LIN {X 0,Y 105.585,Z 420.794,A -85,B 0,C 180,E1 -28240.561,E2 -28240.561} C_VEL
LIN {X 0,Y 105.28,Z 416.678,A -85,B 0,C 180,E1 -28246.489,E2 -28246.489} C_VEL
LIN {X 0,Y 105.21,Z 415.528,A -85,B 0,C 180,E1 -28248.44,E2 -28248.44} C_VEL
LIN {X 0,Y 104.972,Z 413.913,A -85,B 0,C 180,E1 -28252.305,E2 -28252.305} C_VEL
LIN {X 0,Y 105.02,Z 412.014,A -85,B 0,C 180,E1 -28260,E2 -28260} C_VEL
LIN {X 0,Y 104.682,Z 413.549,A -85,B 0,C 180,E1 -28267.965,E2 -28267.965} C_VEL
LIN {X 0,Y 104.931,Z 414.64,A -85,B 0,C 180,E1 -28271.592,E2 -28271.592} C_VEL
LIN {X 0,Y 105.458,Z 417.344,A -85,B 0,C 180,E1 -28277.451,E2 -28277.451} C_VEL
LIN {X 0,Y 106.084,Z 421.23,A -85,B 0,C 180,E1 -28283.422,E2 -28283.422} C_VEL
LIN {X 0,Y 106.272,Z 422.814,A -85,B 0,C 180,E1 -28285.459,E2 -28285.459} C_VEL
LIN {X 0,Y 106.144,Z 427.761,A -85,B 0,C 180,E1 -28290.604,E2 -28290.604} C_VEL
LIN {X 0,Y 105.861,Z 430.108,A -85,B 0,C 180,E1 -28292.818,E2 -28292.818} C_VEL
LIN {X 0,Y 104.957,Z 433.246,A -85,B 0,C 180,E1 -28295.32,E2 -28295.32} C_VEL
LIN {X 0,Y 103.734,Z 435.985,A -85,B 0,C 180,E1 -28297.247,E2 -28297.247} C_VEL
LIN {X 0,Y 96.488,Z 444.212,A -85,B 0,C 180,E1 -28301.708,E2 -28301.708} C_VEL
LIN {X 0,Y 90.783,Z 449.84,A -85,B 0,C 180,E1 -28305.838,E2 -28305.838} C_VEL
LIN {X 0,Y 84.545,Z 455.327,A -85,B 0,C 180,E1 -28311.435,E2 -28311.435} C_VEL
LIN {X 0,Y 79.313,Z 459.625,A -85,B 0,C 180,E1 -28317.885,E2 -28317.885} C_VEL
LIN {X 0,Y 76.364,Z 461.899,A -85,B 0,C 180,E1 -28322.605,E2 -28322.605} C_VEL
LIN {X 0,Y 73.924,Z 463.744,A -85,B 0,C 180,E1 -28327.652,E2 -28327.652} C_VEL
LIN {X 0,Y 70.79,Z 466.108,A -85,B 0,C 180,E1 -28338.55,E2 -28338.55} C_VEL
LIN {X 0,Y 70.624,Z 466.202,A -85,B 0,C 180,E1 -28339.423,E2 -28339.423} C_VEL
LIN {X 0,Y 69.303,Z 466.738,A -85,B 0,C 180,E1 -28344.127,E2 -28344.127} C_VEL
LIN {X 0,Y 66.179,Z 467,A -85,B 0,C 180,E1 -28352.101,E2 -28352.101} C_VEL
LIN {X 0,Y 64.321,Z 466.717,A -85,B 0,C 180,E1 -28358.943,E2 -28358.943} C_VEL
LIN {X 0,Y 64.206,Z 466.166,A -85,B 0,C 180,E1 -28364.243,E2 -28364.243} C_VEL
LIN {X 0,Y 64.524,Z 465.854,A -85,B 0,C 180,E1 -28365.977,E2 -28365.977} C_VEL
LIN {X 0,Y 67.396,Z 464.039,A -85,B 0,C 180,E1 -28374.655,E2 -28374.655} C_VEL
LIN {X 0,Y 71.623,Z 461.169,A -85,B 0,C 180,E1 -28382.664,E2 -28382.664} C_VEL
LIN {X 0,Y 76.993,Z 457.275,A -85,B 0,C 180,E1 -28389.717,E2 -28389.717} C_VEL
LIN {X 0,Y 83.457,Z 452.243,A -85,B 0,C 180,E1 -28395.71,E2 -28395.71} C_VEL
LIN {X 0,Y 90.599,Z 445.904,A -85,B 0,C 180,E1 -28400.873,E2 -28400.873} C_VEL
LIN {X 0,Y 98.238,Z 437.984,A -85,B 0,C 180,E1 -28405.355,E2 -28405.355} C_VEL
LIN {X 0,Y 99.183,Z 436.524,A -85,B 0,C 180,E1 -28406.365,E2 -28406.365} C_VEL
LIN {X 0,Y 99.882,Z 435,A -85,B 0,C 180,E1 -28407.605,E2 -28407.605} C_VEL
LIN {X 0,Y 100.73,Z 431.797,A -85,B 0,C 180,E1 -28410.765,E2 -28410.765} C_VEL
LIN {X 0,Y 101.227,Z 427.772,A -85,B 0,C 180,E1 -28415.382,E2 -28415.382} C_VEL
LIN {X 0,Y 101.117,Z 424.887,A -85,B 0,C 180,E1 -28419.664,E2 -28419.664} C_VEL
LIN {X 0,Y 100.898,Z 422.607,A -85,B 0,C 180,E1 -28423.822,E2 -28423.822} C_VEL
LIN {X 0,Y 100.756,Z 420.842,A -85,B 0,C 180,E1 -28427.921,E2 -28427.921} C_VEL
LIN {X 0,Y 100.642,Z 419.585,A -85,B 0,C 180,E1 -28431.971,E2 -28431.971} C_VEL
LIN {X 0,Y 100.984,Z 418.229,A -85,B 0,C 180,E1 -28440,E2 -28440} C_VEL
LIN {X 0,Y 100.887,Z 420.092,A -85,B 0,C 180,E1 -28448.009,E2 -28448.009} C_VEL
LIN {X 0,Y 100.936,Z 422.857,A -85,B 0,C 180,E1 -28453.899,E2 -28453.899} C_VEL
LIN {X 0,Y 100.864,Z 425.757,A -85,B 0,C 180,E1 -28458.273,E2 -28458.273} C_VEL
LIN {X 0,Y 100.339,Z 430.991,A -85,B 0,C 180,E1 -28464.417,E2 -28464.417} C_VEL
LIN {X 0,Y 99.403,Z 436.189,A -85,B 0,C 180,E1 -28469.664,E2 -28469.664} C_VEL
LIN {X 0,Y 95.514,Z 442.743,A -85,B 0,C 180,E1 -28474.126,E2 -28474.126} C_VEL
LIN {X 0,Y 93.261,Z 445.496,A -85,B 0,C 180,E1 -28475.893,E2 -28475.893} C_VEL
LIN {X 0,Y 85.82,Z 452.677,A -85,B 0,C 180,E1 -28480.754,E2 -28480.754} C_VEL
LIN {X 0,Y 77.996,Z 459.22,A -85,B 0,C 180,E1 -28487.481,E2 -28487.481} C_VEL
LIN {X 0,Y 72.243,Z 463.553,A -85,B 0,C 180,E1 -28494.287,E2 -28494.287} C_VEL
LIN {X 0,Y 69,Z 465.849,A -85,B 0,C 180,E1 -28499.382,E2 -28499.382} C_VEL
LIN {X 0,Y 66.446,Z 467.713,A -85,B 0,C 180,E1 -28504.968,E2 -28504.968} C_VEL
LIN {X 0,Y 63.235,Z 470.118,A -85,B 0,C 180,E1 -28517.154,E2 -28517.154} C_VEL
LIN {X 0,Y 62.585,Z 470.732,A -85,B 0,C 180,E1 -28523.55,E2 -28523.55} C_VEL
LIN {X 0,Y 62.61,Z 470.951,A -85,B 0,C 180,E1 -28529.997,E2 -28529.997} C_VEL
LIN {X 0,Y 62.585,Z 470.716,A -85,B 0,C 180,E1 -28536.445,E2 -28536.445} C_VEL
LIN {X 0,Y 63.234,Z 470.091,A -85,B 0,C 180,E1 -28542.84,E2 -28542.84} C_VEL
LIN {X 0,Y 64.513,Z 469.077,A -85,B 0,C 180,E1 -28549.072,E2 -28549.072} C_VEL
LIN {X 0,Y 66.444,Z 467.659,A -85,B 0,C 180,E1 -28555.027,E2 -28555.027} C_VEL
LIN {X 0,Y 70.563,Z 464.699,A -85,B 0,C 180,E1 -28563.212,E2 -28563.212} C_VEL
LIN {X 0,Y 75.926,Z 460.702,A -85,B 0,C 180,E1 -28570.383,E2 -28570.383} C_VEL
LIN {X 0,Y 83.229,Z 454.761,A -85,B 0,C 180,E1 -28577.284,E2 -28577.284} C_VEL
LIN {X 0,Y 90.652,Z 447.865,A -85,B 0,C 180,E1 -28582.618,E2 -28582.618} C_VEL
LIN {X 0,Y 94.453,Z 443.931,A -85,B 0,C 180,E1 -28584.928,E2 -28584.928} C_VEL
LIN {X 0,Y 98.326,Z 437.876,A -85,B 0,C 180,E1 -28589.055,E2 -28589.055} C_VEL
LIN {X 0,Y 99.315,Z 436.035,A -85,B 0,C 180,E1 -28590.307,E2 -28590.307} C_VEL
LIN {X 0,Y 100.027,Z 432.312,A -85,B 0,C 180,E1 -28593.952,E2 -28593.952} C_VEL
LIN {X 0,Y 100.458,Z 428.924,A -85,B 0,C 180,E1 -28597.597,E2 -28597.597} C_VEL
LIN {X 0,Y 100.743,Z 425.567,A -85,B 0,C 180,E1 -28601.704,E2 -28601.704} C_VEL
LIN {X 0,Y 100.815,Z 421.66,A -85,B 0,C 180,E1 -28607.928,E2 -28607.928} C_VEL
LIN {X 0,Y 100.741,Z 419.889,A -85,B 0,C 180,E1 -28611.98,E2 -28611.98} C_VEL
LIN {X 0,Y 100.924,Z 417.894,A -85,B 0,C 180,E1 -28620,E2 -28620} C_VEL
LIN {X 0,Y 100.487,Z 419.363,A -85,B 0,C 180,E1 -28628.041,E2 -28628.041} C_VEL
LIN {X 0,Y 100.602,Z 420.632,A -85,B 0,C 180,E1 -28632.098,E2 -28632.098} C_VEL
LIN {X 0,Y 100.922,Z 423.386,A -85,B 0,C 180,E1 -28638.263,E2 -28638.263} C_VEL
LIN {X 0,Y 101.083,Z 426.242,A -85,B 0,C 180,E1 -28642.868,E2 -28642.868} C_VEL
LIN {X 0,Y 100.911,Z 429.439,A -85,B 0,C 180,E1 -28646.915,E2 -28646.915} C_VEL
LIN {X 0,Y 100.396,Z 432.935,A -85,B 0,C 180,E1 -28650.746,E2 -28650.746} C_VEL
LIN {X 0,Y 99.186,Z 436.228,A -85,B 0,C 180,E1 -28653.644,E2 -28653.644} C_VEL
LIN {X 0,Y 98.273,Z 437.685,A -85,B 0,C 180,E1 -28654.68,E2 -28654.68} C_VEL
LIN {X 0,Y 90.653,Z 445.655,A -85,B 0,C 180,E1 -28659.176,E2 -28659.176} C_VEL
LIN {X 0,Y 83.507,Z 452.053,A -85,B 0,C 180,E1 -28664.331,E2 -28664.331} C_VEL
LIN {X 0,Y 77.058,Z 457.127,A -85,B 0,C 180,E1 -28670.329,E2 -28670.329} C_VEL
LIN {X 0,Y 71.68,Z 461.059,A -85,B 0,C 180,E1 -28677.37,E2 -28677.37} C_VEL
LIN {X 0,Y 67.406,Z 463.961,A -85,B 0,C 180,E1 -28685.355,E2 -28685.355} C_VEL
LIN {X 0,Y 65.316,Z 465.342,A -85,B 0,C 180,E1 -28691.171,E2 -28691.171} C_VEL
LIN {X 0,Y 63.606,Z 466.441,A -85,B 0,C 180,E1 -28698.488,E2 -28698.488} C_VEL
LIN {X 0,Y 62.755,Z 467.146,A -85,B 0,C 180,E1 -28710.003,E2 -28710.003} C_VEL
LIN {X 0,Y 62.952,Z 466.95,A -85,B 0,C 180,E1 -28716.413,E2 -28716.413} C_VEL
LIN {X 0,Y 64.524,Z 465.854,A -85,B 0,C 180,E1 -28725.977,E2 -28725.977} C_VEL
LIN {X 0,Y 65.342,Z 465.002,A -85,B 0,C 180,E1 -28731.081,E2 -28731.081} C_VEL
LIN {X 0,Y 65.948,Z 463.074,A -85,B 0,C 180,E1 -28739.571,E2 -28739.571} C_VEL
LIN {X 0,Y 67.18,Z 461.056,A -85,B 0,C 180,E1 -28746.126,E2 -28746.126} C_VEL
LIN {X 0,Y 69.265,Z 459.175,A -85,B 0,C 180,E1 -28750.51,E2 -28750.51} C_VEL
LIN {X 0,Y 70.251,Z 458.446,A -85,B 0,C 180,E1 -28751.79,E2 -28751.79} C_VEL
LIN {X 0,Y 78.665,Z 452.457,A -85,B 0,C 180,E1 -28759.413,E2 -28759.413} C_VEL
LIN {X 0,Y 86.287,Z 446.117,A -85,B 0,C 180,E1 -28764.539,E2 -28764.539} C_VEL
LIN {X 0,Y 93.009,Z 439.668,A -85,B 0,C 180,E1 -28768.218,E2 -28768.218} C_VEL
LIN {X 0,Y 94.058,Z 438.215,A -85,B 0,C 180,E1 -28769.233,E2 -28769.233} C_VEL
LIN {X 0,Y 95.177,Z 435.281,A -85,B 0,C 180,E1 -28772.388,E2 -28772.388} C_VEL
LIN {X 0,Y 95.877,Z 432.272,A -85,B 0,C 180,E1 -28776.224,E2 -28776.224} C_VEL
LIN {X 0,Y 95.995,Z 430.765,A -85,B 0,C 180,E1 -28778.527,E2 -28778.527} C_VEL
LIN {X 0,Y 96.055,Z 428.389,A -85,B 0,C 180,E1 -28782.982,E2 -28782.982} C_VEL
LIN {X 0,Y 96.039,Z 426.549,A -85,B 0,C 180,E1 -28787.318,E2 -28787.318} C_VEL
LIN {X 0,Y 96.1,Z 425.235,A -85,B 0,C 180,E1 -28791.589,E2 -28791.589} C_VEL
LIN {X 0,Y 96.563,Z 423.859,A -85,B 0,C 180,E1 -28800,E2 -28800} C_VEL
LIN {X 0,Y 96.326,Z 424.669,A -85,B 0,C 180,E1 -28804.184,E2 -28804.184} C_VEL
LIN {X 0,Y 96.282,Z 425.864,A -85,B 0,C 180,E1 -28808.394,E2 -28808.394} C_VEL
LIN {X 0,Y 96.145,Z 427.688,A -85,B 0,C 180,E1 -28812.667,E2 -28812.667} C_VEL
LIN {X 0,Y 95.774,Z 430.609,A -85,B 0,C 180,E1 -28817.452,E2 -28817.452} C_VEL
LIN {X 0,Y 94.924,Z 434.889,A -85,B 0,C 180,E1 -28822.993,E2 -28822.993} C_VEL
LIN {X 0,Y 94.095,Z 438.07,A -85,B 0,C 180,E1 -28826.625,E2 -28826.625} C_VEL
LIN {X 0,Y 93.37,Z 439.657,A -85,B 0,C 180,E1 -28828.078,E2 -28828.078} C_VEL
LIN {X 0,Y 89.232,Z 445.28,A -85,B 0,C 180,E1 -28832.146,E2 -28832.146} C_VEL
LIN {X 0,Y 81.339,Z 452.462,A -85,B 0,C 180,E1 -28836.941,E2 -28836.941} C_VEL
LIN {X 0,Y 75.244,Z 457.315,A -85,B 0,C 180,E1 -28841.648,E2 -28841.648} C_VEL
LIN {X 0,Y 68.582,Z 462.029,A -85,B 0,C 180,E1 -28848.231,E2 -28848.231} C_VEL
LIN {X 0,Y 62.974,Z 465.634,A -85,B 0,C 180,E1 -28856.079,E2 -28856.079} C_VEL
LIN {X 0,Y 60.046,Z 467.497,A -85,B 0,C 180,E1 -28862.081,E2 -28862.081} C_VEL
LIN {X 0,Y 57.837,Z 468.899,A -85,B 0,C 180,E1 -28868.618,E2 -28868.618} C_VEL
LIN {X 0,Y 56.317,Z 469.902,A -85,B 0,C 180,E1 -28875.544,E2 -28875.544} C_VEL
LIN {X 0,Y 55.54,Z 470.517,A -85,B 0,C 180,E1 -28882.727,E2 -28882.727} C_VEL
LIN {X 0,Y 55.509,Z 470.736,A -85,B 0,C 180,E1 -28889.997,E2 -28889.997} C_VEL
LIN {X 0,Y 55.539,Z 470.5,A -85,B 0,C 180,E1 -28897.266,E2 -28897.266} C_VEL
LIN {X 0,Y 56.315,Z 469.875,A -85,B 0,C 180,E1 -28904.45,E2 -28904.45} C_VEL
LIN {X 0,Y 57.835,Z 468.86,A -85,B 0,C 180,E1 -28911.376,E2 -28911.376} C_VEL
LIN {X 0,Y 60.043,Z 467.442,A -85,B 0,C 180,E1 -28917.913,E2 -28917.913} C_VEL
LIN {X 0,Y 64.724,Z 464.482,A -85,B 0,C 180,E1 -28926.666,E2 -28926.666} C_VEL
LIN {X 0,Y 70.648,Z 460.485,A -85,B 0,C 180,E1 -28934.13,E2 -28934.13} C_VEL
LIN {X 0,Y 77.893,Z 455.091,A -85,B 0,C 180,E1 -28940.609,E2 -28940.609} C_VEL
LIN {X 0,Y 86.502,Z 447.646,A -85,B 0,C 180,E1 -28946.38,E2 -28946.38} C_VEL
LIN {X 0,Y 89.2,Z 445.075,A -85,B 0,C 180,E1 -28947.88,E2 -28947.88} C_VEL
LIN {X 0,Y 93.317,Z 439.465,A -85,B 0,C 180,E1 -28951.922,E2 -28951.922} C_VEL
LIN {X 0,Y 94.117,Z 437.606,A -85,B 0,C 180,E1 -28953.641,E2 -28953.641} C_VEL
LIN {X 0,Y 95.06,Z 433.603,A -85,B 0,C 180,E1 -28958.305,E2 -28958.305} C_VEL
LIN {X 0,Y 95.726,Z 430.132,A -85,B 0,C 180,E1 -28962.922,E2 -28962.922} C_VEL
LIN {X 0,Y 96.017,Z 427.508,A -85,B 0,C 180,E1 -28967.315,E2 -28967.315} C_VEL
LIN {X 0,Y 96.162,Z 425.655,A -85,B 0,C 180,E1 -28971.595,E2 -28971.595} C_VEL
LIN {X 0,Y 96.225,Z 424.422,A -85,B 0,C 180,E1 -28975.812,E2 -28975.812} C_VEL
LIN {X 0,Y 96.517,Z 423.536,A -85,B 0,C 180,E1 -28980,E2 -28980} C_VEL
LIN {X 0,Y 95.947,Z 425.044,A -85,B 0,C 180,E1 -28988.424,E2 -28988.424} C_VEL
LIN {X 0,Y 95.912,Z 426.328,A -85,B 0,C 180,E1 -28992.699,E2 -28992.699} C_VEL
LIN {X 0,Y 95.974,Z 429.117,A -85,B 0,C 180,E1 -28999.018,E2 -28999.018} C_VEL
LIN {X 0,Y 95.757,Z 432.06,A -85,B 0,C 180,E1 -29003.808,E2 -29003.808} C_VEL
LIN {X 0,Y 95.126,Z 434.969,A -85,B 0,C 180,E1 -29007.561,E2 -29007.561} C_VEL
LIN {X 0,Y 94.705,Z 436.493,A -85,B 0,C 180,E1 -29009.323,E2 -29009.323} C_VEL
LIN {X 0,Y 94.055,Z 437.924,A -85,B 0,C 180,E1 -29010.771,E2 -29010.771} C_VEL
LIN {X 0,Y 93.043,Z 439.38,A -85,B 0,C 180,E1 -29011.823,E2 -29011.823} C_VEL
LIN {X 0,Y 85.048,Z 447.033,A -85,B 0,C 180,E1 -29016.327,E2 -29016.327} C_VEL
LIN {X 0,Y 76.307,Z 454.074,A -85,B 0,C 180,E1 -29022.544,E2 -29022.544} C_VEL
LIN {X 0,Y 69.669,Z 458.756,A -85,B 0,C 180,E1 -29029.032,E2 -29029.032} C_VEL
LIN {X 0,Y 64.072,Z 462.333,A -85,B 0,C 180,E1 -29036.744,E2 -29036.744} C_VEL
LIN {X 0,Y 61.027,Z 464.177,A -85,B 0,C 180,E1 -29042.575,E2 -29042.575} C_VEL
LIN {X 0,Y 58.634,Z 465.558,A -85,B 0,C 180,E1 -29048.929,E2 -29048.929} C_VEL
LIN {X 0,Y 56.927,Z 466.54,A -85,B 0,C 180,E1 -29055.709,E2 -29055.709} C_VEL
LIN {X 0,Y 55.671,Z 467.361,A -85,B 0,C 180,E1 -29070.003,E2 -29070.003} C_VEL
LIN {X 0,Y 55.92,Z 467.165,A -85,B 0,C 180,E1 -29077.223,E2 -29077.223} C_VEL
LIN {X 0,Y 57.623,Z 466.127,A -85,B 0,C 180,E1 -29087.514,E2 -29087.514} C_VEL
LIN {X 0,Y 61.015,Z 464.253,A -85,B 0,C 180,E1 -29097.437,E2 -29097.437} C_VEL
LIN {X 0,Y 65.755,Z 461.384,A -85,B 0,C 180,E1 -29106.007,E2 -29106.007} C_VEL
LIN {X 0,Y 70.251,Z 458.446,A -85,B 0,C 180,E1 -29111.79,E2 -29111.79} C_VEL
LIN {X 0,Y 73.05,Z 456.216,A -85,B 0,C 180,E1 -29115.557,E2 -29115.557} C_VEL
LIN {X 0,Y 76.861,Z 452.182,A -85,B 0,C 180,E1 -29121.862,E2 -29121.862} C_VEL
LIN {X 0,Y 81.242,Z 447.528,A -85,B 0,C 180,E1 -29127.366,E2 -29127.366} C_VEL
LIN {X 0,Y 84.73,Z 444.272,A -85,B 0,C 180,E1 -29129.795,E2 -29129.795} C_VEL
LIN {X 0,Y 88.036,Z 441.237,A -85,B 0,C 180,E1 -29131.421,E2 -29131.421} C_VEL
LIN {X 0,Y 89.108,Z 439.823,A -85,B 0,C 180,E1 -29132.684,E2 -29132.684} C_VEL
LIN {X 0,Y 90.314,Z 436.591,A -85,B 0,C 180,E1 -29137.102,E2 -29137.102} C_VEL
LIN {X 0,Y 90.779,Z 433.928,A -85,B 0,C 180,E1 -29141.96,E2 -29141.96} C_VEL
LIN {X 0,Y 90.981,Z 432.024,A -85,B 0,C 180,E1 -29146.6,E2 -29146.6} C_VEL
LIN {X 0,Y 91.175,Z 430.632,A -85,B 0,C 180,E1 -29151.131,E2 -29151.131} C_VEL
LIN {X 0,Y 91.507,Z 429.598,A -85,B 0,C 180,E1 -29156.807,E2 -29156.807} C_VEL
LIN {X 0,Y 91.845,Z 429.233,A -85,B 0,C 180,E1 -29160,E2 -29160} C_VEL
LIN {X 0,Y 91.535,Z 430.065,A -85,B 0,C 180,E1 -29164.403,E2 -29164.403} C_VEL
LIN {X 0,Y 91.154,Z 432.227,A -85,B 0,C 180,E1 -29171.113,E2 -29171.113} C_VEL
LIN {X 0,Y 90.648,Z 434.644,A -85,B 0,C 180,E1 -29175.745,E2 -29175.745} C_VEL
LIN {X 0,Y 89.379,Z 438.718,A -85,B 0,C 180,E1 -29181.607,E2 -29181.607} C_VEL
LIN {X 0,Y 88.28,Z 441.474,A -85,B 0,C 180,E1 -29185.018,E2 -29185.018} C_VEL
LIN {X 0,Y 85.479,Z 445.055,A -85,B 0,C 180,E1 -29187.886,E2 -29187.886} C_VEL
LIN {X 0,Y 82.814,Z 447.619,A -85,B 0,C 180,E1 -29189.554,E2 -29189.554} C_VEL
LIN {X 0,Y 74.429,Z 454.377,A -85,B 0,C 180,E1 -29194.51,E2 -29194.51} C_VEL
LIN {X 0,Y 65.73,Z 460.377,A -85,B 0,C 180,E1 -29201.54,E2 -29201.54} C_VEL
LIN {X 0,Y 59.174,Z 464.345,A -85,B 0,C 180,E1 -29209.212,E2 -29209.212} C_VEL
LIN {X 0,Y 53.836,Z 467.281,A -85,B 0,C 180,E1 -29218.519,E2 -29218.519} C_VEL
LIN {X 0,Y 49.467,Z 469.687,A -85,B 0,C 180,E1 -29233.488,E2 -29233.488} C_VEL
LIN {X 0,Y 48.497,Z 470.302,A -85,B 0,C 180,E1 -29241.664,E2 -29241.664} C_VEL
LIN {X 0,Y 48.427,Z 470.521,A -85,B 0,C 180,E1 -29249.996,E2 -29249.996} C_VEL
LIN {X 0,Y 48.496,Z 470.284,A -85,B 0,C 180,E1 -29258.329,E2 -29258.329} C_VEL
LIN {X 0,Y 49.465,Z 469.659,A -85,B 0,C 180,E1 -29266.505,E2 -29266.505} C_VEL
LIN {X 0,Y 51.248,Z 468.643,A -85,B 0,C 180,E1 -29274.289,E2 -29274.289} C_VEL
LIN {X 0,Y 53.833,Z 467.224,A -85,B 0,C 180,E1 -29281.476,E2 -29281.476} C_VEL
LIN {X 0,Y 59.17,Z 464.265,A -85,B 0,C 180,E1 -29290.784,E2 -29290.784} C_VEL
LIN {X 0,Y 65.724,Z 460.267,A -85,B 0,C 180,E1 -29298.457,E2 -29298.457} C_VEL
LIN {X 0,Y 74.36,Z 454.268,A -85,B 0,C 180,E1 -29305.454,E2 -29305.454} C_VEL
LIN {X 0,Y 82.771,Z 447.428,A -85,B 0,C 180,E1 -29310.489,E2 -29310.489} C_VEL
LIN {X 0,Y 85.44,Z 444.844,A -85,B 0,C 180,E1 -29312.153,E2 -29312.153} C_VEL
LIN {X 0,Y 88.214,Z 441.319,A -85,B 0,C 180,E1 -29314.929,E2 -29314.929} C_VEL
LIN {X 0,Y 89.684,Z 437.26,A -85,B 0,C 180,E1 -29320.104,E2 -29320.104} C_VEL
LIN {X 0,Y 90.589,Z 434.147,A -85,B 0,C 180,E1 -29324.849,E2 -29324.849} C_VEL
LIN {X 0,Y 91.034,Z 432.053,A -85,B 0,C 180,E1 -29328.872,E2 -29328.872} C_VEL
LIN {X 0,Y 91.186,Z 431.16,A -85,B 0,C 180,E1 -29331.133,E2 -29331.133} C_VEL
LIN {X 0,Y 91.521,Z 429.594,A -85,B 0,C 180,E1 -29336.589,E2 -29336.589} C_VEL
LIN {X 0,Y 91.814,Z 428.923,A -85,B 0,C 180,E1 -29340,E2 -29340} C_VEL
LIN {X 0,Y 91.037,Z 430.448,A -85,B 0,C 180,E1 -29348.882,E2 -29348.882} C_VEL
LIN {X 0,Y 90.879,Z 431.799,A -85,B 0,C 180,E1 -29353.415,E2 -29353.415} C_VEL
LIN {X 0,Y 90.744,Z 433.654,A -85,B 0,C 180,E1 -29358.047,E2 -29358.047} C_VEL
LIN {X 0,Y 90.219,Z 436.382,A -85,B 0,C 180,E1 -29362.924,E2 -29362.924} C_VEL
LIN {X 0,Y 89.013,Z 439.744,A -85,B 0,C 180,E1 -29367.562,E2 -29367.562} C_VEL
LIN {X 0,Y 88.076,Z 440.972,A -85,B 0,C 180,E1 -29368.635,E2 -29368.635} C_VEL
LIN {X 0,Y 79.69,Z 448.359,A -85,B 0,C 180,E1 -29373.095,E2 -29373.095} C_VEL
LIN {X 0,Y 71.689,Z 454.291,A -85,B 0,C 180,E1 -29378.352,E2 -29378.352} C_VEL
LIN {X 0,Y 64.458,Z 458.973,A -85,B 0,C 180,E1 -29384.875,E2 -29384.875} C_VEL
LIN {X 0,Y 58.254,Z 462.549,A -85,B 0,C 180,E1 -29392.904,E2 -29392.904} C_VEL
LIN {X 0,Y 54.83,Z 464.393,A -85,B 0,C 180,E1 -29399.16,E2 -29399.16} C_VEL
LIN {X 0,Y 52.076,Z 465.774,A -85,B 0,C 180,E1 -29406.121,E2 -29406.121} C_VEL
LIN {X 0,Y 50.085,Z 466.756,A -85,B 0,C 180,E1 -29413.705,E2 -29413.705} C_VEL
LIN {X 0,Y 48.581,Z 467.577,A -85,B 0,C 180,E1 -29430.004,E2 -29430.004} C_VEL
LIN {X 0,Y 48.885,Z 467.38,A -85,B 0,C 180,E1 -29438.269,E2 -29438.269} C_VEL
LIN {X 0,Y 50.086,Z 466.793,A -85,B 0,C 180,E1 -29446.302,E2 -29446.302} C_VEL
LIN {X 0,Y 54.817,Z 464.468,A -85,B 0,C 180,E1 -29460.856,E2 -29460.856} C_VEL
LIN {X 0,Y 60.155,Z 461.598,A -85,B 0,C 180,E1 -29469.987,E2 -29469.987} C_VEL
LIN {X 0,Y 66.683,Z 457.704,A -85,B 0,C 180,E1 -29477.544,E2 -29477.544} C_VEL
LIN {X 0,Y 74.244,Z 452.67,A -85,B 0,C 180,E1 -29483.576,E2 -29483.576} C_VEL
LIN {X 0,Y 82.368,Z 446.331,A -85,B 0,C 180,E1 -29488.569,E2 -29488.569} C_VEL
LIN {X 0,Y 84.73,Z 444.272,A -85,B 0,C 180,E1 -29489.795,E2 -29489.795} C_VEL
LIN {X 0,Y 85.953,Z 442.94,A -85,B 0,C 180,E1 -29490.916,E2 -29490.916} C_VEL
LIN {X 0,Y 86.622,Z 441.391,A -85,B 0,C 180,E1 -29493.19,E2 -29493.19} C_VEL
LIN {X 0,Y 86.42,Z 440.352,A -85,B 0,C 180,E1 -29495.719,E2 -29495.719} C_VEL
LIN {X 0,Y 85.262,Z 438.124,A -85,B 0,C 180,E1 -29503.569,E2 -29503.569} C_VEL
LIN {X 0,Y 85.826,Z 436.126,A -85,B 0,C 180,E1 -29509.314,E2 -29509.314} C_VEL
LIN {X 0,Y 86.279,Z 434.86,A -85,B 0,C 180,E1 -29515.327,E2 -29515.327} C_VEL
LIN {X 0,Y 86.813,Z 434.311,A -85,B 0,C 180,E1 -29520,E2 -29520} C_VEL
LIN {X 0,Y 86.366,Z 435.2,A -85,B 0,C 180,E1 -29524.667,E2 -29524.667} C_VEL
LIN {X 0,Y 85.841,Z 437.082,A -85,B 0,C 180,E1 -29530.738,E2 -29530.738} C_VEL
LIN {X 0,Y 85.292,Z 438.748,A -85,B 0,C 180,E1 -29534.312,E2 -29534.312} C_VEL
LIN {X 0,Y 83.883,Z 442.007,A -85,B 0,C 180,E1 -29539.581,E2 -29539.581} C_VEL
LIN {X 0,Y 83.159,Z 443.421,A -85,B 0,C 180,E1 -29541.619,E2 -29541.619} C_VEL
LIN {X 0,Y 82.159,Z 444.824,A -85,B 0,C 180,E1 -29543.133,E2 -29543.133} C_VEL
LIN {X 0,Y 79.538,Z 447.404,A -85,B 0,C 180,E1 -29545.081,E2 -29545.081} C_VEL
LIN {X 0,Y 69.862,Z 454.709,A -85,B 0,C 180,E1 -29550.198,E2 -29550.198} C_VEL
LIN {X 0,Y 61.243,Z 460.163,A -85,B 0,C 180,E1 -29556.551,E2 -29556.551} C_VEL
LIN {X 0,Y 53.97,Z 464.129,A -85,B 0,C 180,E1 -29564.253,E2 -29564.253} C_VEL
LIN {X 0,Y 47.891,Z 467.065,A -85,B 0,C 180,E1 -29574.052,E2 -29574.052} C_VEL
LIN {X 0,Y 42.676,Z 469.471,A -85,B 0,C 180,E1 -29590.766,E2 -29590.766} C_VEL
LIN {X 0,Y 41.471,Z 470.086,A -85,B 0,C 180,E1 -29600.239,E2 -29600.239} C_VEL
LIN {X 0,Y 41.327,Z 470.305,A -85,B 0,C 180,E1 -29609.996,E2 -29609.996} C_VEL
LIN {X 0,Y 41.47,Z 470.068,A -85,B 0,C 180,E1 -29619.753,E2 -29619.753} C_VEL
LIN {X 0,Y 42.674,Z 469.442,A -85,B 0,C 180,E1 -29629.227,E2 -29629.227} C_VEL
LIN {X 0,Y 44.834,Z 468.426,A -85,B 0,C 180,E1 -29638.047,E2 -29638.047} C_VEL
LIN {X 0,Y 47.888,Z 467.007,A -85,B 0,C 180,E1 -29645.942,E2 -29645.942} C_VEL
LIN {X 0,Y 53.965,Z 464.047,A -85,B 0,C 180,E1 -29655.742,E2 -29655.742} C_VEL
LIN {X 0,Y 61.237,Z 460.05,A -85,B 0,C 180,E1 -29663.447,E2 -29663.447} C_VEL
LIN {X 0,Y 69.933,Z 454.503,A -85,B 0,C 180,E1 -29669.836,E2 -29669.836} C_VEL
LIN {X 0,Y 79.494,Z 447.209,A -85,B 0,C 180,E1 -29674.978,E2 -29674.978} C_VEL
LIN {X 0,Y 82.133,Z 444.609,A -85,B 0,C 180,E1 -29676.898,E2 -29676.898} C_VEL
LIN {X 0,Y 83.112,Z 443.203,A -85,B 0,C 180,E1 -29678.452,E2 -29678.452} C_VEL
LIN {X 0,Y 84.492,Z 440.141,A -85,B 0,C 180,E1 -29683.075,E2 -29683.075} C_VEL
LIN {X 0,Y 85.131,Z 438.642,A -85,B 0,C 180,E1 -29685.661,E2 -29685.661} C_VEL
LIN {X 0,Y 85.89,Z 436.383,A -85,B 0,C 180,E1 -29690.581,E2 -29690.581} C_VEL
LIN {X 0,Y 86.291,Z 434.988,A -85,B 0,C 180,E1 -29695.329,E2 -29695.329} C_VEL
LIN {X 0,Y 86.799,Z 434.037,A -85,B 0,C 180,E1 -29700,E2 -29700} C_VEL
LIN {X 0,Y 85.859,Z 435.3,A -85,B 0,C 180,E1 -29707.904,E2 -29707.904} C_VEL
LIN {X 0,Y 85.475,Z 437.044,A -85,B 0,C 180,E1 -29714.281,E2 -29714.281} C_VEL
LIN {X 0,Y 85.34,Z 437.882,A -85,B 0,C 180,E1 -29716.753,E2 -29716.753} C_VEL
LIN {X 0,Y 84.727,Z 439.914,A -85,B 0,C 180,E1 -29720.99,E2 -29720.99} C_VEL
LIN {X 0,Y 83.595,Z 442.308,A -85,B 0,C 180,E1 -29724.858,E2 -29724.858} C_VEL
LIN {X 0,Y 74.61,Z 449.685,A -85,B 0,C 180,E1 -29729.395,E2 -29729.395} C_VEL
LIN {X 0,Y 67.511,Z 454.509,A -85,B 0,C 180,E1 -29733.617,E2 -29733.617} C_VEL
LIN {X 0,Y 59.65,Z 459.191,A -85,B 0,C 180,E1 -29740.025,E2 -29740.025} C_VEL
LIN {X 0,Y 52.761,Z 462.766,A -85,B 0,C 180,E1 -29748.245,E2 -29748.245} C_VEL
LIN {X 0,Y 48.856,Z 464.609,A -85,B 0,C 180,E1 -29754.878,E2 -29754.878} C_VEL
LIN {X 0,Y 43.334,Z 466.971,A -85,B 0,C 180,E1 -29771.078,E2 -29771.078} C_VEL
LIN {X 0,Y 41.481,Z 467.792,A -85,B 0,C 180,E1 -29790.004,E2 -29790.004} C_VEL
LIN {X 0,Y 41.888,Z 467.595,A -85,B 0,C 180,E1 -29799.663,E2 -29799.663} C_VEL
LIN {X 0,Y 43.336,Z 467.008,A -85,B 0,C 180,E1 -29808.93,E2 -29808.93} C_VEL
LIN {X 0,Y 48.843,Z 464.683,A -85,B 0,C 180,E1 -29825.143,E2 -29825.143} C_VEL
LIN {X 0,Y 54.906,Z 461.813,A -85,B 0,C 180,E1 -29834.753,E2 -29834.753} C_VEL
LIN {X 0,Y 62.113,Z 457.918,A -85,B 0,C 180,E1 -29842.38,E2 -29842.38} C_VEL
LIN {X 0,Y 70.264,Z 452.884,A -85,B 0,C 180,E1 -29848.235,E2 -29848.235} C_VEL
LIN {X 0,Y 78.898,Z 446.544,A -85,B 0,C 180,E1 -29852.973,E2 -29852.973} C_VEL
LIN {X 0,Y 83.617,Z 442.551,A -85,B 0,C 180,E1 -29855.149,E2 -29855.149} C_VEL
LIN {X 0,Y 84.791,Z 440.203,A -85,B 0,C 180,E1 -29858.861,E2 -29858.861} C_VEL
LIN {X 0,Y 85.079,Z 439.255,A -85,B 0,C 180,E1 -29860.705,E2 -29860.705} C_VEL
LIN {X 0,Y 85.262,Z 438.124,A -85,B 0,C 180,E1 -29863.569,E2 -29863.569} C_VEL
LIN {X 0,Y 84.964,Z 437.63,A -85,B 0,C 180,E1 -29866.166,E2 -29866.166} C_VEL
LIN {X 0,Y 83.546,Z 438.055,A -85,B 0,C 180,E1 -29869.64,E2 -29869.64} C_VEL
LIN {X 0,Y 81.319,Z 439.28,A -85,B 0,C 180,E1 -29875.09,E2 -29875.09} C_VEL
LIN {X 0,Y 81.147,Z 439.339,A -85,B 0,C 180,E1 -29877.969,E2 -29877.969} C_VEL
LIN {X 0,Y 81.474,Z 439.106,A -85,B 0,C 180,E1 -29880,E2 -29880} C_VEL
LIN {X 0,Y 80.898,Z 440.062,A -85,B 0,C 180,E1 -29884.984,E2 -29884.984} C_VEL
LIN {X 0,Y 80.304,Z 441.559,A -85,B 0,C 180,E1 -29890.08,E2 -29890.08} C_VEL
LIN {X 0,Y 79.521,Z 443.06,A -85,B 0,C 180,E1 -29893.543,E2 -29893.543} C_VEL
LIN {X 0,Y 77.856,Z 445.906,A -85,B 0,C 180,E1 -29898.586,E2 -29898.586} C_VEL
LIN {X 0,Y 76.709,Z 447.183,A -85,B 0,C 180,E1 -29900.096,E2 -29900.096} C_VEL
LIN {X 0,Y 69.051,Z 452.839,A -85,B 0,C 180,E1 -29903.645,E2 -29903.645} C_VEL
LIN {X 0,Y 60.168,Z 458.361,A -85,B 0,C 180,E1 -29908.827,E2 -29908.827} C_VEL
LIN {X 0,Y 51.845,Z 462.692,A -85,B 0,C 180,E1 -29915.571,E2 -29915.571} C_VEL
LIN {X 0,Y 46.804,Z 464.989,A -85,B 0,C 180,E1 -29921.336,E2 -29921.336} C_VEL
LIN {X 0,Y 42.32,Z 466.849,A -85,B 0,C 180,E1 -29928.369,E2 -29928.369} C_VEL
LIN {X 0,Y 36.027,Z 469.255,A -85,B 0,C 180,E1 -29947.031,E2 -29947.031} C_VEL
LIN {X 0,Y 34.493,Z 469.871,A -85,B 0,C 180,E1 -29958.238,E2 -29958.238} C_VEL
LIN {X 0,Y 34.242,Z 470.09,A -85,B 0,C 180,E1 -29969.995,E2 -29969.995} C_VEL
LIN {X 0,Y 34.491,Z 469.852,A -85,B 0,C 180,E1 -29981.751,E2 -29981.751} C_VEL
LIN {X 0,Y 36.025,Z 469.225,A -85,B 0,C 180,E1 -29992.96,E2 -29992.96} C_VEL
LIN {X 0,Y 38.684,Z 468.209,A -85,B 0,C 180,E1 -30003.021,E2 -30003.021} C_VEL
LIN {X 0,Y 42.316,Z 466.789,A -85,B 0,C 180,E1 -30011.625,E2 -30011.625} C_VEL
LIN {X 0,Y 49.254,Z 463.83,A -85,B 0,C 180,E1 -30021.694,E2 -30021.694} C_VEL
LIN {X 0,Y 57.287,Z 459.833,A -85,B 0,C 180,E1 -30029.17,E2 -30029.17} C_VEL
LIN {X 0,Y 67.462,Z 453.724,A -85,B 0,C 180,E1 -30035.595,E2 -30035.595} C_VEL
LIN {X 0,Y 76.679,Z 446.987,A -85,B 0,C 180,E1 -30039.944,E2 -30039.944} C_VEL
LIN {X 0,Y 77.814,Z 445.71,A -85,B 0,C 180,E1 -30041.477,E2 -30041.477} C_VEL
LIN {X 0,Y 79.454,Z 442.83,A -85,B 0,C 180,E1 -30046.638,E2 -30046.638} C_VEL
LIN {X 0,Y 80.176,Z 441.42,A -85,B 0,C 180,E1 -30049.903,E2 -30049.903} C_VEL
LIN {X 0,Y 80.82,Z 439.871,A -85,B 0,C 180,E1 -30055.012,E2 -30055.012} C_VEL
LIN {X 0,Y 81.457,Z 438.858,A -85,B 0,C 180,E1 -30060,E2 -30060} C_VEL
LIN {X 0,Y 80.438,Z 439.997,A -85,B 0,C 180,E1 -30067.665,E2 -30067.665} C_VEL
LIN {X 0,Y 80.287,Z 440.464,A -85,B 0,C 180,E1 -30070.083,E2 -30070.083} C_VEL
LIN {X 0,Y 79.777,Z 441.9,A -85,B 0,C 180,E1 -30075.325,E2 -30075.325} C_VEL
LIN {X 0,Y 79.354,Z 442.944,A -85,B 0,C 180,E1 -30078.058,E2 -30078.058} C_VEL
LIN {X 0,Y 78.591,Z 444.366,A -85,B 0,C 180,E1 -30080.959,E2 -30080.959} C_VEL
LIN {X 0,Y 77.371,Z 445.42,A -85,B 0,C 180,E1 -30081.751,E2 -30081.751} C_VEL
LIN {X 0,Y 69.845,Z 450.926,A -85,B 0,C 180,E1 -30085.103,E2 -30085.103} C_VEL
LIN {X 0,Y 60.948,Z 456.411,A -85,B 0,C 180,E1 -30090.143,E2 -30090.143} C_VEL
LIN {X 0,Y 52.685,Z 460.711,A -85,B 0,C 180,E1 -30096.841,E2 -30096.841} C_VEL
LIN {X 0,Y 47.701,Z 462.982,A -85,B 0,C 180,E1 -30102.558,E2 -30102.558} C_VEL
LIN {X 0,Y 43.237,Z 464.826,A -85,B 0,C 180,E1 -30109.451,E2 -30109.451} C_VEL
LIN {X 0,Y 36.694,Z 467.187,A -85,B 0,C 180,E1 -30127.483,E2 -30127.483} C_VEL
LIN {X 0,Y 34.4,Z 468.007,A -85,B 0,C 180,E1 -30150.005,E2 -30150.005} C_VEL
LIN {X 0,Y 34.92,Z 467.81,A -85,B 0,C 180,E1 -30161.616,E2 -30161.616} C_VEL
LIN {X 0,Y 36.696,Z 467.223,A -85,B 0,C 180,E1 -30172.527,E2 -30172.527} C_VEL
LIN {X 0,Y 43.224,Z 464.898,A -85,B 0,C 180,E1 -30190.575,E2 -30190.575} C_VEL
LIN {X 0,Y 50.115,Z 462.027,A -85,B 0,C 180,E1 -30200.476,E2 -30200.476} C_VEL
LIN {X 0,Y 58.056,Z 458.132,A -85,B 0,C 180,E1 -30207.933,E2 -30207.933} C_VEL
LIN {X 0,Y 66.803,Z 453.098,A -85,B 0,C 180,E1 -30213.414,E2 -30213.414} C_VEL
LIN {X 0,Y 75.937,Z 446.758,A -85,B 0,C 180,E1 -30217.748,E2 -30217.748} C_VEL
LIN {X 0,Y 78.629,Z 444.571,A -85,B 0,C 180,E1 -30219.051,E2 -30219.051} C_VEL
LIN {X 0,Y 79.405,Z 443.157,A -85,B 0,C 180,E1 -30221.954,E2 -30221.954} C_VEL
LIN {X 0,Y 80.393,Z 440.641,A -85,B 0,C 180,E1 -30229.93,E2 -30229.93} C_VEL
LIN {X 0,Y 80.857,Z 439.675,A -85,B 0,C 180,E1 -30235.013,E2 -30235.013} C_VEL
LIN {X 0,Y 81.147,Z 439.339,A -85,B 0,C 180,E1 -30237.969,E2 -30237.969} C_VEL
LIN {X 0,Y 80.952,Z 439.562,A -85,B 0,C 180,E1 -30240.213,E2 -30240.213} C_VEL
LIN {X 0,Y 79.568,Z 440.952,A -85,B 0,C 180,E1 -30243.173,E2 -30243.173} C_VEL
LIN {X 0,Y 73.753,Z 446.724,A -85,B 0,C 180,E1 -30251.748,E2 -30251.748} C_VEL
LIN {X 0,Y 72.7,Z 448.181,A -85,B 0,C 180,E1 -30254.821,E2 -30254.821} C_VEL
LIN {X 0,Y 71.355,Z 449.366,A -85,B 0,C 180,E1 -30256.19,E2 -30256.19} C_VEL
LIN {X 0,Y 60.148,Z 456.452,A -85,B 0,C 180,E1 -30260.805,E2 -30260.805} C_VEL
LIN {X 0,Y 50.965,Z 461.167,A -85,B 0,C 180,E1 -30266.313,E2 -30266.313} C_VEL
LIN {X 0,Y 42.427,Z 464.773,A -85,B 0,C 180,E1 -30274.076,E2 -30274.076} C_VEL
LIN {X 0,Y 37.289,Z 466.633,A -85,B 0,C 180,E1 -30281.065,E2 -30281.065} C_VEL
LIN {X 0,Y 29.608,Z 469.039,A -85,B 0,C 180,E1 -30301.652,E2 -30301.652} C_VEL
LIN {X 0,Y 27.562,Z 469.655,A -85,B 0,C 180,E1 -30315.221,E2 -30315.221} C_VEL
LIN {X 0,Y 27.129,Z 469.874,A -85,B 0,C 180,E1 -30329.993,E2 -30329.993} C_VEL
LIN {X 0,Y 27.56,Z 469.636,A -85,B 0,C 180,E1 -30344.767,E2 -30344.767} C_VEL
LIN {X 0,Y 29.605,Z 469.009,A -85,B 0,C 180,E1 -30358.337,E2 -30358.337} C_VEL
LIN {X 0,Y 32.939,Z 467.992,A -85,B 0,C 180,E1 -30369.791,E2 -30369.791} C_VEL
LIN {X 0,Y 37.284,Z 466.572,A -85,B 0,C 180,E1 -30378.929,E2 -30378.929} C_VEL
LIN {X 0,Y 45.184,Z 463.613,A -85,B 0,C 180,E1 -30388.804,E2 -30388.804} C_VEL
LIN {X 0,Y 53.987,Z 459.616,A -85,B 0,C 180,E1 -30395.668,E2 -30395.668} C_VEL
LIN {X 0,Y 63.529,Z 454.341,A -85,B 0,C 180,E1 -30400.763,E2 -30400.763} C_VEL
LIN {X 0,Y 71.324,Z 449.182,A -85,B 0,C 180,E1 -30403.876,E2 -30403.876} C_VEL
LIN {X 0,Y 72.664,Z 447.976,A -85,B 0,C 180,E1 -30405.27,E2 -30405.27} C_VEL
LIN {X 0,Y 73.954,Z 446.208,A -85,B 0,C 180,E1 -30409.044,E2 -30409.044} C_VEL
LIN {X 0,Y 75.04,Z 444.48,A -85,B 0,C 180,E1 -30414.626,E2 -30414.626} C_VEL
LIN {X 0,Y 75.845,Z 443.391,A -85,B 0,C 180,E1 -30420,E2 -30420} C_VEL
LIN {X 0,Y 74.782,Z 444.352,A -85,B 0,C 180,E1 -30427.223,E2 -30427.223} C_VEL
LIN {X 0,Y 74.412,Z 445.019,A -85,B 0,C 180,E1 -30430.889,E2 -30430.889} C_VEL
LIN {X 0,Y 73.459,Z 446.755,A -85,B 0,C 180,E1 -30436.929,E2 -30436.929} C_VEL
LIN {X 0,Y 72.368,Z 447.613,A -85,B 0,C 180,E1 -30437.602,E2 -30437.602} C_VEL
LIN {X 0,Y 63.963,Z 453.138,A -85,B 0,C 180,E1 -30440.952,E2 -30440.952} C_VEL
LIN {X 0,Y 54.646,Z 458.211,A -85,B 0,C 180,E1 -30445.817,E2 -30445.817} C_VEL
LIN {X 0,Y 45.957,Z 462.141,A -85,B 0,C 180,E1 -30452.753,E2 -30452.753} C_VEL
LIN {X 0,Y 38.123,Z 465.042,A -85,B 0,C 180,E1 -30462.498,E2 -30462.498} C_VEL
LIN {X 0,Y 33.718,Z 466.422,A -85,B 0,C 180,E1 -30471.303,E2 -30471.303} C_VEL
LIN {X 0,Y 30.254,Z 467.403,A -85,B 0,C 180,E1 -30482.323,E2 -30482.323} C_VEL
LIN {X 0,Y 27.302,Z 468.222,A -85,B 0,C 180,E1 -30510.006,E2 -30510.006} C_VEL
LIN {X 0,Y 28,Z 468.025,A -85,B 0,C 180,E1 -30524.543,E2 -30524.543} C_VEL
LIN {X 0,Y 30.256,Z 467.438,A -85,B 0,C 180,E1 -30537.688,E2 -30537.688} C_VEL
LIN {X 0,Y 38.112,Z 465.113,A -85,B 0,C 180,E1 -30557.534,E2 -30557.534} C_VEL
LIN {X 0,Y 45.911,Z 462.243,A -85,B 0,C 180,E1 -30567.351,E2 -30567.351} C_VEL
LIN {X 0,Y 54.623,Z 458.346,A -85,B 0,C 180,E1 -30574.247,E2 -30574.247} C_VEL
LIN {X 0,Y 63.945,Z 453.311,A -85,B 0,C 180,E1 -30579.106,E2 -30579.106} C_VEL
LIN {X 0,Y 72.36,Z 447.809,A -85,B 0,C 180,E1 -30582.478,E2 -30582.478} C_VEL
LIN {X 0,Y 73.49,Z 446.976,A -85,B 0,C 180,E1 -30583.006,E2 -30583.006} C_VEL
LIN {X 0,Y 74.431,Z 445.231,A -85,B 0,C 180,E1 -30589.114,E2 -30589.114} C_VEL
LIN {X 0,Y 75.168,Z 444.193,A -85,B 0,C 180,E1 -30594.635,E2 -30594.635} C_VEL
LIN {X 0,Y 75.86,Z 443.618,A -85,B 0,C 180,E1 -30600,E2 -30600} C_VEL
LIN {X 0,Y 75.123,Z 444.65,A -85,B 0,C 180,E1 -30605.368,E2 -30605.368} C_VEL
LIN {X 0,Y 74.071,Z 446.333,A -85,B 0,C 180,E1 -30610.939,E2 -30610.939} C_VEL
LIN {X 0,Y 73.753,Z 446.724,A -85,B 0,C 180,E1 -30611.748,E2 -30611.748} C_VEL
LIN {X 0,Y 72.579,Z 447.843,A -85,B 0,C 180,E1 -30613.154,E2 -30613.154} C_VEL
LIN {X 0,Y 70.258,Z 449.548,A -85,B 0,C 180,E1 -30614.159,E2 -30614.159} C_VEL
LIN {X 0,Y 66.324,Z 451.969,A -85,B 0,C 180,E1 -30614.562,E2 -30614.562} C_VEL
LIN {X 0,Y 58.303,Z 456.129,A -85,B 0,C 180,E1 -30614.463,E2 -30614.463} C_VEL
LIN {X 0,Y 55.727,Z 457.41,A -85,B 0,C 180,E1 -30615.145,E2 -30615.145} C_VEL
LIN {X 0,Y 45.053,Z 462.26,A -85,B 0,C 180,E1 -30620.609,E2 -30620.609} C_VEL
LIN {X 0,Y 38.883,Z 464.557,A -85,B 0,C 180,E1 -30625.337,E2 -30625.337} C_VEL
LIN {X 0,Y 33.042,Z 466.417,A -85,B 0,C 180,E1 -30631.692,E2 -30631.692} C_VEL
LIN {X 0,Y 27.849,Z 467.819,A -85,B 0,C 180,E1 -30640.784,E2 -30640.784} C_VEL
LIN {X 0,Y 20.77,Z 469.439,A -85,B 0,C 180,E1 -30670.214,E2 -30670.214} C_VEL
LIN {X 0,Y 20.022,Z 469.659,A -85,B 0,C 180,E1 -30689.991,E2 -30689.991} C_VEL
LIN {X 0,Y 20.768,Z 469.42,A -85,B 0,C 180,E1 -30709.77,E2 -30709.77} C_VEL
LIN {X 0,Y 27.844,Z 467.776,A -85,B 0,C 180,E1 -30739.208,E2 -30739.208} C_VEL
LIN {X 0,Y 33.036,Z 466.355,A -85,B 0,C 180,E1 -30748.302,E2 -30748.302} C_VEL
LIN {X 0,Y 41.937,Z 463.395,A -85,B 0,C 180,E1 -30757.164,E2 -30757.164} C_VEL
LIN {X 0,Y 51.465,Z 459.399,A -85,B 0,C 180,E1 -30762.908,E2 -30762.908} C_VEL
LIN {X 0,Y 62.972,Z 453.255,A -85,B 0,C 180,E1 -30767.54,E2 -30767.54} C_VEL
LIN {X 0,Y 67.377,Z 450.496,A -85,B 0,C 180,E1 -30768.915,E2 -30768.915} C_VEL
LIN {X 0,Y 68.266,Z 449.533,A -85,B 0,C 180,E1 -30771.422,E2 -30771.422} C_VEL
LIN {X 0,Y 68.823,Z 448.826,A -85,B 0,C 180,E1 -30774.139,E2 -30774.139} C_VEL
LIN {X 0,Y 69.964,Z 447.628,A -85,B 0,C 180,E1 -30780,E2 -30780} C_VEL
LIN {X 0,Y 68.957,Z 448.336,A -85,B 0,C 180,E1 -30786.434,E2 -30786.434} C_VEL
LIN {X 0,Y 68.117,Z 449.331,A -85,B 0,C 180,E1 -30791.909,E2 -30791.909} C_VEL
LIN {X 0,Y 67.014,Z 450.181,A -85,B 0,C 180,E1 -30793.154,E2 -30793.154} C_VEL
LIN {X 0,Y 58.477,Z 455.159,A -85,B 0,C 180,E1 -30795.97,E2 -30795.97} C_VEL
LIN {X 0,Y 48.759,Z 459.841,A -85,B 0,C 180,E1 -30800.477,E2 -30800.477} C_VEL
LIN {X 0,Y 39.516,Z 463.414,A -85,B 0,C 180,E1 -30807.232,E2 -30807.232} C_VEL
LIN {X 0,Y 33.74,Z 465.258,A -85,B 0,C 180,E1 -30813.583,E2 -30813.583} C_VEL
LIN {X 0,Y 24.199,Z 467.618,A -85,B 0,C 180,E1 -30834.499,E2 -30834.499} C_VEL
LIN {X 0,Y 20.22,Z 468.437,A -85,B 0,C 180,E1 -30870.009,E2 -30870.009} C_VEL
LIN {X 0,Y 21.208,Z 468.24,A -85,B 0,C 180,E1 -30889.362,E2 -30889.362} C_VEL
LIN {X 0,Y 24.201,Z 467.653,A -85,B 0,C 180,E1 -30905.515,E2 -30905.515} C_VEL
LIN {X 0,Y 33.732,Z 465.328,A -85,B 0,C 180,E1 -30926.456,E2 -30926.456} C_VEL
LIN {X 0,Y 42.496,Z 462.458,A -85,B 0,C 180,E1 -30935.456,E2 -30935.456} C_VEL
LIN {X 0,Y 51.938,Z 458.56,A -85,B 0,C 180,E1 -30941.305,E2 -30941.305} C_VEL
LIN {X 0,Y 61.772,Z 453.525,A -85,B 0,C 180,E1 -30945.261,E2 -30945.261} C_VEL
LIN {X 0,Y 67.023,Z 450.364,A -85,B 0,C 180,E1 -30946.948,E2 -30946.948} C_VEL
LIN {X 0,Y 68.144,Z 449.517,A -85,B 0,C 180,E1 -30948.096,E2 -30948.096} C_VEL
LIN {X 0,Y 69.143,Z 448.391,A -85,B 0,C 180,E1 -30954.166,E2 -30954.166} C_VEL
LIN {X 0,Y 69.973,Z 447.834,A -85,B 0,C 180,E1 -30960,E2 -30960} C_VEL
LIN {X 0,Y 68.922,Z 448.955,A -85,B 0,C 180,E1 -30965.852,E2 -30965.852} C_VEL
LIN {X 0,Y 67.984,Z 450.053,A -85,B 0,C 180,E1 -30969.578,E2 -30969.578} C_VEL
LIN {X 0,Y 67.475,Z 450.622,A -85,B 0,C 180,E1 -30971.079,E2 -30971.079} C_VEL
LIN {X 0,Y 57.999,Z 456.237,A -85,B 0,C 180,E1 -30974.205,E2 -30974.205} C_VEL
LIN {X 0,Y 55.727,Z 457.41,A -85,B 0,C 180,E1 -30975.145,E2 -30975.145} C_VEL
LIN {X 0,Y 50.538,Z 459.842,A -85,B 0,C 180,E1 -30976.742,E2 -30976.742} C_VEL
LIN {X 0,Y 41.229,Z 463.19,A -85,B 0,C 180,E1 -30977.866,E2 -30977.866} C_VEL
LIN {X 0,Y 31.711,Z 465.796,A -85,B 0,C 180,E1 -30979.769,E2 -30979.769} C_VEL
LIN {X 0,Y 26.337,Z 467.009,A -85,B 0,C 180,E1 -30983.981,E2 -30983.981} C_VEL
LIN {X 0,Y 18.354,Z 468.607,A -85,B 0,C 180,E1 -31000.005,E2 -31000.005} C_VEL
LIN {X 0,Y 14.275,Z 469.223,A -85,B 0,C 180,E1 -31020.492,E2 -31020.492} C_VEL
LIN {X 0,Y 12.929,Z 469.443,A -85,B 0,C 180,E1 -31049.986,E2 -31049.986} C_VEL
LIN {X 0,Y 14.272,Z 469.204,A -85,B 0,C 180,E1 -31079.487,E2 -31079.487} C_VEL
LIN {X 0,Y 18.349,Z 468.576,A -85,B 0,C 180,E1 -31099.982,E2 -31099.982} C_VEL
LIN {X 0,Y 23.805,Z 467.559,A -85,B 0,C 180,E1 -31112.321,E2 -31112.321} C_VEL
LIN {X 0,Y 29.91,Z 466.137,A -85,B 0,C 180,E1 -31120.013,E2 -31120.013} C_VEL
LIN {X 0,Y 39.718,Z 463.178,A -85,B 0,C 180,E1 -31126.685,E2 -31126.685} C_VEL
LIN {X 0,Y 49.839,Z 459.181,A -85,B 0,C 180,E1 -31130.757,E2 -31130.757} C_VEL
LIN {X 0,Y 62.054,Z 452.9,A -85,B 0,C 180,E1 -31134.088,E2 -31134.088} C_VEL
LIN {X 0,Y 63.289,Z 451.902,A -85,B 0,C 180,E1 -31137.93,E2 -31137.93} C_VEL
LIN {X 0,Y 63.75,Z 451.544,A -85,B 0,C 180,E1 -31140,E2 -31140} C_VEL
LIN {X 0,Y 62.74,Z 452.134,A -85,B 0,C 180,E1 -31146.432,E2 -31146.432} C_VEL
LIN {X 0,Y 59.923,Z 453.808,A -85,B 0,C 180,E1 -31148.381,E2 -31148.381} C_VEL
LIN {X 0,Y 50.124,Z 458.643,A -85,B 0,C 180,E1 -31151.069,E2 -31151.069} C_VEL
LIN {X 0,Y 40.084,Z 462.575,A -85,B 0,C 180,E1 -31155.37,E2 -31155.37} C_VEL
LIN {X 0,Y 30.393,Z 465.474,A -85,B 0,C 180,E1 -31162.356,E2 -31162.356} C_VEL
LIN {X 0,Y 18.885,Z 467.834,A -85,B 0,C 180,E1 -31181.918,E2 -31181.918} C_VEL
LIN {X 0,Y 13.132,Z 468.653,A -85,B 0,C 180,E1 -31230.013,E2 -31230.013} C_VEL
LIN {X 0,Y 14.714,Z 468.455,A -85,B 0,C 180,E1 -31258.544,E2 -31258.544} C_VEL
LIN {X 0,Y 18.889,Z 467.868,A -85,B 0,C 180,E1 -31278.098,E2 -31278.098} C_VEL
LIN {X 0,Y 30.389,Z 465.543,A -85,B 0,C 180,E1 -31297.693,E2 -31297.693} C_VEL
LIN {X 0,Y 40.068,Z 462.673,A -85,B 0,C 180,E1 -31304.744,E2 -31304.744} C_VEL
LIN {X 0,Y 50.119,Z 458.773,A -85,B 0,C 180,E1 -31309,E2 -31309} C_VEL
LIN {X 0,Y 59.944,Z 453.957,A -85,B 0,C 180,E1 -31311.686,E2 -31311.686} C_VEL
LIN {X 0,Y 62.796,Z 452.283,A -85,B 0,C 180,E1 -31313.574,E2 -31313.574} C_VEL
LIN {X 0,Y 63.776,Z 451.706,A -85,B 0,C 180,E1 -31320,E2 -31320} C_VEL
LIN {X 0,Y 62.98,Z 452.399,A -85,B 0,C 180,E1 -31324.21,E2 -31324.21} C_VEL
LIN {X 0,Y 60.112,Z 454.202,A -85,B 0,C 180,E1 -31326.404,E2 -31326.404} C_VEL
LIN {X 0,Y 49.845,Z 459.304,A -85,B 0,C 180,E1 -31329.244,E2 -31329.244} C_VEL
LIN {X 0,Y 39.724,Z 463.268,A -85,B 0,C 180,E1 -31333.314,E2 -31333.314} C_VEL
LIN {X 0,Y 29.916,Z 466.201,A -85,B 0,C 180,E1 -31339.982,E2 -31339.982} C_VEL
LIN {X 0,Y 26.337,Z 467.009,A -85,B 0,C 180,E1 -31343.981,E2 -31343.981} C_VEL
LIN {X 0,Y 21.157,Z 468.049,A -85,B 0,C 180,E1 -31350.469,E2 -31350.469} C_VEL
LIN {X 0,Y 15.793,Z 468.784,A -85,B 0,C 180,E1 -31358.208,E2 -31358.208} C_VEL
LIN {X 0,Y 6.771,Z 469.359,A -85,B 0,C 180,E1 -31403.267,E2 -31403.267} C_VEL
LIN {X 0,Y 8.852,Z 468.983,A -85,B 0,C 180,E1 -31463.16,E2 -31463.16} C_VEL
LIN {X 0,Y 14.813,Z 468.359,A -85,B 0,C 180,E1 -31481.567,E2 -31481.567} C_VEL
LIN {X 0,Y 28.278,Z 465.92,A -85,B 0,C 180,E1 -31493.718,E2 -31493.718} C_VEL
LIN {X 0,Y 38.703,Z 462.961,A -85,B 0,C 180,E1 -31497.007,E2 -31497.007} C_VEL
LIN {X 0,Y 51.636,Z 457.854,A -85,B 0,C 180,E1 -31499.411,E2 -31499.411} C_VEL
LIN {X 0,Y 56.22,Z 455.651,A -85,B 0,C 180,E1 -31500,E2 -31500} C_VEL
LIN {X 0,Y 57.335,Z 455.056,A -85,B 0,C 180,E1 -31500.788,E2 -31500.788} C_VEL
LIN {X 0,Y 56.252,Z 455.592,A -85,B 0,C 180,E1 -31501.954,E2 -31501.954} C_VEL
LIN {X 0,Y 45.765,Z 460.275,A -85,B 0,C 180,E1 -31503.541,E2 -31503.541} C_VEL
LIN {X 0,Y 35.348,Z 463.848,A -85,B 0,C 180,E1 -31506.28,E2 -31506.28} C_VEL
LIN {X 0,Y 28.458,Z 465.691,A -85,B 0,C 180,E1 -31508.987,E2 -31508.987} C_VEL
LIN {X 0,Y 15.095,Z 468.05,A -85,B 0,C 180,E1 -31521.42,E2 -31521.42} C_VEL
LIN {X 0,Y 6.033,Z 468.868,A -85,B 0,C 180,E1 -31590.029,E2 -31590.029} C_VEL
LIN {X 0,Y 9.134,Z 468.67,A -85,B 0,C 180,E1 -31640.329,E2 -31640.329} C_VEL
LIN {X 0,Y 15.1,Z 468.083,A -85,B 0,C 180,E1 -31658.594,E2 -31658.594} C_VEL
LIN {X 0,Y 28.459,Z 465.758,A -85,B 0,C 180,E1 -31671.073,E2 -31671.073} C_VEL
LIN {X 0,Y 38.809,Z 462.887,A -85,B 0,C 180,E1 -31674.917,E2 -31674.917} C_VEL
LIN {X 0,Y 51.682,Z 457.914,A -85,B 0,C 180,E1 -31677.535,E2 -31677.535} C_VEL
LIN {X 0,Y 56.256,Z 455.752,A -85,B 0,C 180,E1 -31678.114,E2 -31678.114} C_VEL
LIN {X 0,Y 57.336,Z 455.213,A -85,B 0,C 180,E1 -31679.083,E2 -31679.083} C_VEL
LIN {X 0,Y 56.226,Z 455.808,A -85,B 0,C 180,E1 -31680,E2 -31680} C_VEL
LIN {X 0,Y 45.701,Z 460.523,A -85,B 0,C 180,E1 -31681.548,E2 -31681.548} C_VEL
LIN {X 0,Y 35.224,Z 464.127,A -85,B 0,C 180,E1 -31683.893,E2 -31683.893} C_VEL
LIN {X 0,Y 23.523,Z 466.958,A -85,B 0,C 180,E1 -31688.95,E2 -31688.95} C_VEL
LIN {X 0,Y 14.818,Z 468.392,A -85,B 0,C 180,E1 -31698.425,E2 -31698.425} C_VEL
LIN {X 0,Y 8.813,Z 469.008,A -85,B 0,C 180,E1 -31717.078,E2 -31717.078} C_VEL
LIN {X 0,Y 5.824,Z 469.228,A -85,B 0,C 180,E1 -31769.97,E2 -31769.97} C_VEL
LIN {X 0,Y 8.852,Z 468.983,A -85,B 0,C 180,E1 -31823.16,E2 -31823.16} C_VEL
LIN {X 0,Y 10.572,Z 470.975,A -85,B 0,C 180,E1 -31831.075,E2 -31831.075} C_VEL
LIN {X 0,Y 10.572,Z 600,A -85,B 0,C 180,E1 -31831.075,E2 -31831.075} C_VEL
LIN {X 0,Y 10.572,Z 600,A -85,B 0,C 180,E1 -31831.075,E2 -31831.075}

QRS_NEXT_CUT()

QRS_NEXT()
QRS_HOME()

END
